(* PLC project 117_1_V0.5.project, CODESYS CODESYS V3.5 SP17 Patch 3 *)
(* stored: creationDateTime 1970-01-01T00:00:00, modificationDateTime 2026-03-26T18:14:32.4070562 *)

TYPE ALL_AI : (tenza1000kgSensor, tenza50kgSensor, motionSensor, lastAnalogInIndex);
END_TYPE
